FUNCTION_BLOCK FB_AlarmSystem

VAR_INPUT			// Input variables
	ClearButton : BOOL;
	EmergencyButton : BOOL;
END_VAR

VAR					// Internal (instance) variables
	bIsInitialized : BOOL;
	latch : BOOL := FALSE;
END_VAR

IF (NOT bIsInitialized) THEN	// Initialization, since functions can't run in top pane
	bIsInitialized := TRUE;
	gAL.fbAlarm.CreateEx(TC_Events.TankAlarmEvent.Emergency, TRUE, 0);
END_IF

IF ( (NOT EmergencyButton) AND (NOT latch) ) THEN
	gAL.fbAlarm.Raise(0); // 0 -> Current time
	latch := TRUE;
END_IF

IF (ClearButton AND gAL.fbAlarm.bRaised) THEN
	gAL.fbAlarm.Clear(0, TRUE);	// .Clear(CurrentTime, ConfirmAlarm)
	latch := FALSE;
END_IF

END_FUNCTION_BLOCK

(* stored: Version 1.1.0.1, ProductVersion 3.1.4024.12
   POU FB_AlarmSystem: Id {ff8af221-7c2c-420a-82d2-c72830098d6c}, SpecialFunc None *)
